TYPE ST_ServiceExecutionSnapshot :
STRUCT
	Valid : BOOL;
	ServiceId : UDINT;
	ResponseId : UDINT;
	PackMLOut : ST_PML_Base_Out;
	ExecuteSubState : UDINT;
	CompletionBehavior : E_ServiceCompletionBehavior;
END_STRUCT
END_TYPE

(* stored: Version 1.1.0.1, ProductVersion 3.1.4026.18
   DUT ST_ServiceExecutionSnapshot: Id {911dfa98-9995-4fc5-9896-9e719d59ee89} *)
